FUNCTION_BLOCK NullImageSerializer IMPLEMENTS I_ImageSerializer
VAR
END_VAR

METHOD PUBLIC ConnectTo
VAR_INPUT
	ImageSerializer : I_ImageSerializer;
END_VAR
END_METHOD

METHOD PUBLIC GetTotalSerializablePixelCount : UDINT
VAR_INPUT
END_VAR
GetTotalSerializablePixelCount := 0;
END_METHOD

PROPERTY PUBLIC PixelCount : UDINT
GET
PixelCount := 0;
END_GET
END_PROPERTY

METHOD PUBLIC TryGetPixel : BOOL
VAR_INPUT
	PixelIndex : UDINT;
	Reader : I_PixelReader;
END_VAR
TryGetPixel := FALSE;
END_METHOD

METHOD PUBLIC UpdateImage
VAR_INPUT
	Source : ITcVnImage;
END_VAR
END_METHOD

END_FUNCTION_BLOCK

(* stored: Version 1.1.0.1, ProductVersion 3.1.4024.13
   POU NullImageSerializer: Id {2a0e6b0d-b602-4b71-9152-c6f55d4baf8e}, SpecialFunc None
   Method ConnectTo: Id {abec6695-355a-4221-bb10-54168c04ab50}
   Method GetTotalSerializablePixelCount: Id {d402f688-098f-4de0-8b0e-c25b3509152e}
   Property PixelCount: Id {7d567119-b3da-4b6c-acba-ef6349c8663c}
   Get Get: Id {435eb4e0-3cd6-4977-891c-6680cd3733d7}
   Method TryGetPixel: Id {f7ba1710-8e4e-4b6b-be1b-ca79db67a3b7}
   Method UpdateImage: Id {77b43070-e487-48b4-ae21-9746621f679a} *)
